// TIA Portal V16 export
// export: Created 2024-12-03T15:41:41.1940093Z, ExportSetting WithDefaults, DisplayName Totally Integrated Automation Portal, DisplayVersion V16 Update 6, DisplayName TIA Portal Version Control Interface, DisplayVersion V16 Update 2, DisplayName TIA Portal Openness, DisplayVersion V16 Update 6, DisplayName TIA Portal Teamcenter Gateway, DisplayVersion V16, DisplayName SINAMICS Startdrive Advanced, DisplayVersion V16 Update 5, DisplayName SINAMICS Startdrive G130, G150, S120, S150, SINAMICS MV, S210, DisplayVersion V16 Update 5, DisplayName SINAMICS Startdrive G110M, G120, G120C, G120D, G120P, G115D, DisplayVersion V16 Update 5, DisplayName STEP 7 Professional, DisplayVersion V16 Update 6, DisplayName STEP 7 Safety, DisplayVersion V16, DisplayName WinCC Advanced / Unified PC, DisplayVersion V16 Update 6
FUNCTION_BLOCK "StepperControllerSimple"   // FB110, SCL
{ S7_Optimized_Access := 'FALSE' }
VERSION : 0.1
// stored: AutoNumber true, IsIECCheckEnabled false, SetENOAutomatically false, UDAEnableTagReadback false
   VAR_INPUT
      I_StepNumber : DInt;
      I_NextStepNumber : DInt;
      I_Condition : Bool;
      I_ConditionTime : Time;
   END_VAR
   VAR_OUTPUT
      O_ConditionTrans : Bool;
   END_VAR
   VAR_IN_OUT
      IO_StepNumber : DInt;
      IO_PrevStepNumber : DInt;
   END_VAR
   VAR DB_SPECIFIC
      conditionTime : TON_TIME;
   END_VAR
   VAR_TEMP
      T_Bug : Bool;
   END_VAR
BEGIN
   //Reset flags
   #O_ConditionTrans := false;

   IF #I_StepNumber = #IO_StepNumber THEN

       IF #I_Condition THEN
           IF #I_ConditionTime = t#0ms THEN
               "SetPrevStepNumber_FC"(I_Step := #IO_StepNumber,
                                      IO_PrevStep := #IO_PrevStepNumber);
               #IO_StepNumber := #I_NextStepNumber;
               #O_ConditionTrans := true;
           ELSE
               #conditionTime(IN := #I_Condition,
                              Q => #T_Bug,
                              PT := #I_ConditionTime);

               IF #conditionTime.Q THEN
                   "SetPrevStepNumber_FC"(I_Step := #IO_StepNumber,
                                          IO_PrevStep := #IO_PrevStepNumber);
                   #IO_StepNumber := #I_NextStepNumber;
                   #O_ConditionTrans := true;
               END_IF;
           END_IF;
       END_IF;
   ELSE
       RESET_TIMER(#conditionTime);
       #O_ConditionTrans := FALSE;

   END_IF;
END_FUNCTION_BLOCK
